// TwinCAT 3 PLC project Untitled1
// ProgramVersion: 3.1.4024.0
// libraries:
//   Tc2_HVAC, * (Beckhoff Automation GmbH)
//   Tc2_Standard, * (Beckhoff Automation GmbH)
//   Tc2_System, * (Beckhoff Automation GmbH)
//   Tc2_SystemC69xx, * (Beckhoff Automation GmbH)
//   Tc3_Module, * (Beckhoff Automation GmbH)
//   Util, * (System)
//   VisuSymbols,3.5.10.0,System
// project tree:
//   / GlobalTextList.TcGTLO, PlcTask.TcTTO, Visualization Manager.TcVMO (not stored)
//   GVLs/ GVL.TcGVL
//   POUs/FunctionBlocks/ Start_Stop.TcPOU, Trapizoidal.TcPOU
//   POUs/Functions/ ScaleOutput.TcPOU
//   POUs/ MAIN.TcPOU
//   POUs/Programs/ Motor_Control.TcPOU, ProgramSequence.TcPOU, Reset.TcPOU
//   VISUs/ Visualization.TcVIS
// real-time tasks:
//   TASK PlcTask: cycle T#10ms, priority 20, ADS port 350

CONFIGURATION Untitled1
    RESOURCE PLC ON TwinCAT3
        TASK PlcTask(INTERVAL := T#10ms, PRIORITY := 20);
        PROGRAM MAIN WITH PlcTask : MAIN;
    END_RESOURCE
END_CONFIGURATION

// ---- GVLs/GVL.TcGVL
{attribute 'qualified_only'}
VAR_GLOBAL
	(*Digital Input*)
	SART_STOP AT %IX0.0 : BOOL;		 	 (*To Start And To Stop System*)
	EM_STOP AT %IX0.1 : BOOL; 			 (*To Turn Power Of The System*)
	Conveyor2_Free AT %IX0.2 : BOOL;	 (*When The Conveyor2 is free*)
	Reset_Count AT %IX0.3 : BOOL;  		 (*Reset the Product counter value*)
	
	(*Analog Inputs*) (*Hiervoor vanwege gemak gebruik gemaakt van 0,1,3 normaal zou dit hogere waarde zijn wat uitgelezen wordt*)
	SensorInput AT %IW100 : INT;		 (*Noting=0 Red=1 Blue=2 Collor detection sensor*)

	(*Digital Output*)
	Motor1_State AT %QX10.0 : BOOL; 	 (*To indicate if the morot is on or of (1=on 0=of)*)
	Motor2_State AT %QX10.1 : BOOL;		 (*To indicate if the morot is on or of (1=on 0=of)*)
	
	(*Analog Output*)
	Motor1_Speed AT %QW200 : DINT;		 (*The Motor 1 Speed Output 0-65535*)
	Motor2_Speed AT %QW201 : DINT;		 (*The Motor 2 Speed Output 0-65535*)
	
	(*System Variables*)
	SystemState : INT; 					 (*System State 0=OFF 1=ON 2=EM_STOP*)	
	System_Start_Stop : BOOL;			 (*GVL Start/Stop variable 0=stop 1=start*)
	ProductA_Amount : INT;				 (*Amount of products counted*)
	ProductB_Amount : INT;				 (*Amount of products counted*)
	
	(*Motor Variables*)
	SetMotor1_Speed : INT;				 (*Set The Motor Speed in the program from hmi km/h*)
	SetMotor2_Speed : INT; 				 (*Set The Motor Speed in the program from hmi km/h*)
	CurrentMotor1_Speed : INT;			 (*The current speed after Trapizoidal function*)
	CurrentMotor2_Speed : INT;			 (*The current speed after Trapizoidal function*)
	Motor2_DirectionL : BOOL;			 (*Determine Motor direction*)
	Motor2_DirectionR : BOOL;			 (*Determine Motor direct*)

	

END_VAR

// ---- POUs/MAIN.TcPOU
PROGRAM MAIN
VAR
END_VAR

(*Calling Different Programs*)
Motor_Control ();
ProgramSequence ();
Reset ();

END_PROGRAM

// ---- POUs/Programs/Motor_Control.TcPOU
PROGRAM Motor_Control
VAR
	Start_Stop_0: Start_Stop;
	Trapizoidal_0: Trapizoidal;
	Trapizoidal_1: Trapizoidal;
	BLINK_0: BLINK;
	R_TRIG_0: R_TRIG;
	
	Timer : BOOL;
END_VAR

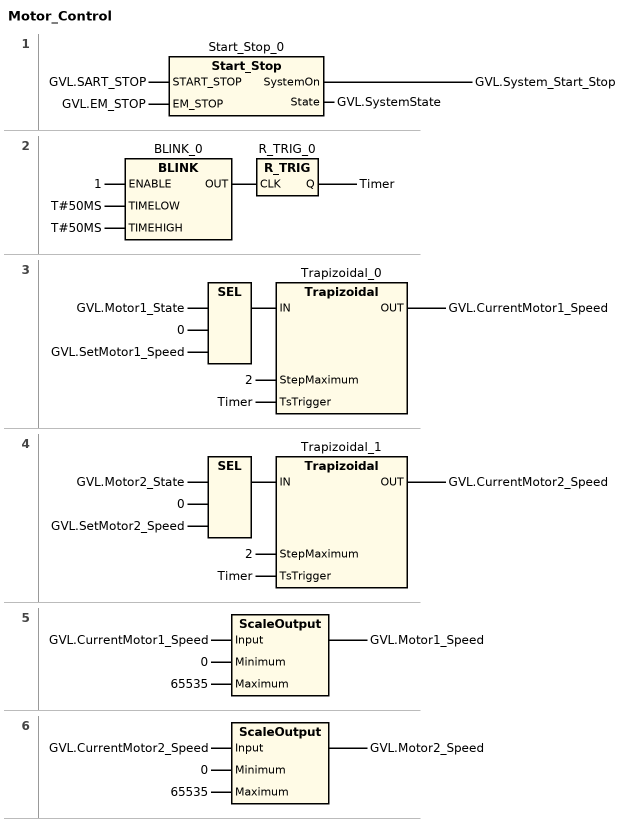
// NETWORK 1
Start_Stop_0(START_STOP := GVL.SART_STOP, EM_STOP := GVL.EM_STOP, State => GVL.SystemState); // Start_Stop
GVL.System_Start_Stop := Start_Stop_0.SystemOn;

// NETWORK 2
BLINK_0(ENABLE := 1, TIMELOW := T#50MS, TIMEHIGH := T#50MS); // BLINK
R_TRIG_0(CLK := BLINK_0.OUT); // R_TRIG
Timer := R_TRIG_0.Q;

// NETWORK 3
Trapizoidal_0(IN := SEL(GVL.Motor1_State, 0, GVL.SetMotor1_Speed), StepMaximum := 2, TsTrigger := Timer); // Trapizoidal
GVL.CurrentMotor1_Speed := Trapizoidal_0.OUT;

// NETWORK 4
Trapizoidal_1(IN := SEL(GVL.Motor2_State, 0, GVL.SetMotor2_Speed), StepMaximum := 2, TsTrigger := Timer); // Trapizoidal
GVL.CurrentMotor2_Speed := Trapizoidal_1.OUT;

// NETWORK 5
GVL.Motor1_Speed := ScaleOutput(Input := GVL.CurrentMotor1_Speed, Minimum := 0, Maximum := 65535);

// NETWORK 6
GVL.Motor2_Speed := ScaleOutput(Input := GVL.CurrentMotor2_Speed, Minimum := 0, Maximum := 65535);

END_PROGRAM

// ---- POUs/FunctionBlocks/Start_Stop.TcPOU
(*Vincent Molenkamp : 519540*)
FUNCTION_BLOCK Start_Stop
VAR_INPUT
	START_STOP : BOOL;
	EM_STOP : BOOL;
END_VAR
VAR_OUTPUT
	SystemOn : BOOL;
	State : INT;
END_VAR

VAR
	X: INT;
END_VAR

CASE X OF
	0: IF START_STOP THEN
		SystemOn := 1;
		X := 1;
		END_IF;
	1: IF NOT START_STOP THEN
			X := 2;
			State := 1;
		END_IF;
	2: IF START_STOP THEN
		SystemOn := 0;
		X := 3;
		END_IF;	
	3: IF NOT START_STOP THEN
		X := 0;	
		State := 0;
		END_IF;
	END_CASE
	
	IF NOT EM_STOP THEN
	X := 4;
	SystemOn := 0;
	State := 2;
	END_IF; 
	
	IF X = 4 AND EM_STOP AND NOT START_STOP THEN
		X := 0;
	END_IF

END_FUNCTION_BLOCK

// ---- POUs/FunctionBlocks/Trapizoidal.TcPOU
(*Vincent Molenkamp : 519540*)
FUNCTION_BLOCK Trapizoidal
(*Function Block To slowly increase speed*)
VAR_INPUT
	IN: INT;
	StepMaximum: INT;
	TsTrigger: BOOL;
END_VAR

VAR_OUTPUT	
	OUT: INT;
END_VAR

VAR
	Y_1: INT;
	Y_0: INT;
END_VAR

IF TsTrigger = 1 THEN
Y_1 := Y_0; (*De waarde van de vorige cicle in Y_1 Zetten*)

(*Wanneer de waarde van de voorige cicle lager is als de waarde van de nieuwe dan + 1 tot hij gelijk is*)
IF Y_1 < IN THEN
	Y_0 := 	Y_1 + StepMaximum;
END_IF

(*Wanneer de waarde van de voorige cicle Hoger is als de waarde van de nieuwe dan - 1 tot hij gelijk is*)
IF Y_1 > IN THEN
	Y_0 := Y_1 - StepMaximum;
END_IF

(*De output waarde meegeven*)
OUT := Y_0;
END_IF

END_FUNCTION_BLOCK

// ---- POUs/Functions/ScaleOutput.TcPOU
(*Vincent Molenkamp : 519540*)
FUNCTION ScaleOutput : DINT
(*Om de output waarde te scalen naar Van DINT naar WORD*)
VAR_INPUT	
	Input: INT;	  (*waarde die gescaled moet worden*)
	Minimum: INT; (*De minimum input waarde*)
	Maximum: INT; (*De maximum input waarde*)
END_VAR
VAR
	X: DINT;
END_VAR

(* To set minimum and maximum values for the input *)
IF Input < Minimum THEN
	Input := Minimum;
ELSIF Input > Maximum THEN
	Input := Maximum;
END_IF

(* Calculating the output value does not work with negative minimum *) 
ScaleOutput := ((Input-Minimum)*65535)/(Maximum-Minimum);

END_FUNCTION

// ---- POUs/Programs/ProgramSequence.TcPOU
PROGRAM ProgramSequence
VAR
	X: INT;
END_VAR

IF NOT GVL.System_Start_Stop THEN
	X := 10;
	GVL.Motor1_State := 0;
	GVL.Motor2_State := 0;	
END_IF

	CASE X OF
0: IF NOT GVL.Motor1_State THEN
 	GVL.Motor1_State := 1;
	X := 1;
	END_IF
	
1: IF GVL.SensorInput = 1 THEN
	GVL.Motor2_Direction := 0;
	GVL.Motor2_State := 1;
	GVL.ProductA_Amount := GVL.ProductA_Amount + 1;
	X := 2;
	ELSIF GVL.SensorInput = 2 THEN
	GVL.Motor2_Direction := 1;
	GVL.Motor2_State := 1;
	X := 2;
	GVL.ProductB_Amount := GVL.ProductB_Amount + 1;
	END_IF
	
2: 	GVL.Motor1_State := 0;
	IF GVL.Conveyor2_Free THEN
	X := 0;
	END_IF
	END_CASE

END_PROGRAM

// ---- POUs/Programs/Reset.TcPOU
PROGRAM Reset
(*What happens when reset is pressed*)
VAR
END_VAR

IF GVL.Reset_Count THEN
	GVL.ProductA_Amount := 0; (*To Reset Product Count*)
	GVL.ProductB_Amount := 0; (*To Reset Product Count*)
END_IF

END_PROGRAM

// ---- GlobalTextList.TcGTLO
TEXTLIST GlobalTextList
  21 = 'Amount A:%i'
  901 = 'Amount B:%i'
  356 = 'Conveyor 2 Free'
  483 = 'EM_Stop'
  0 = 'Motor 1'
  269 = 'Motor 1 Speed'
  816 = 'Motor 2'
  610 = 'Motor 2 Speed'
  52 = 'Product Type'
  237 = 'Reset Count'
  958 = 'Sensors'
  700 = 'Set Motor 1 Speed:%i'
  46 = 'Start/Stop'
  395 = 'Start_Stop Button'
  487 = 'System State:%i'
END_TEXTLIST

// ---- VISUs/Visualization.TcVIS
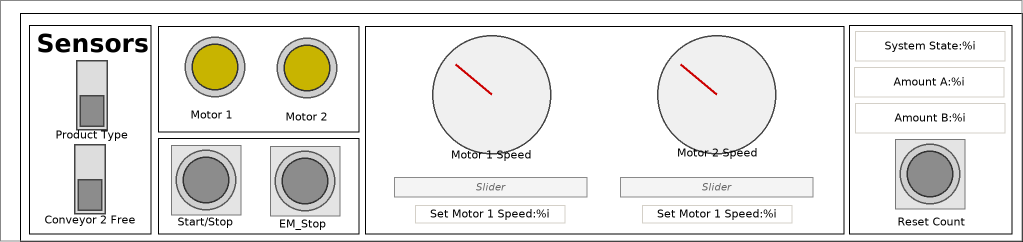
VISUALIZATION Visualization  // 1023x242
    Rectangle (20,13 1003x229)
    Rectangle (849,25 163x209)
    Rectangle (158,138 201x96)
    Rectangle (365,26 479x208)
    Rectangle (158,26 201x106)
    Rectangle (29,25 122x209)
    Lamp1 (180,32 70x70), style: Lamp-Lamp1-Yellow
    Lamp1 (272,33 70x70), variable: GVL.Motor2_State, style: Lamp-Lamp1-Yellow
    DipSwitch (57,60 70x70), variable: GVL.SensorInput, behaviour: TOGGLE, style: Switch-DipSwitch-Gray
    DipSwitch (55,144 70x70), variable: GVL.Conveyor2_Free, behaviour: TOGGLE, style: Switch-DipSwitch-Gray
    Label (18,28 150x30), "Sensors"
    Label (176,100 71x30), "Motor 1"
    Label (271,102 71x30), "Motor 2"
    Meter180 (386,35 211x119), value: GVL.CurrentMotor1_Speed, style: Meter-Meter180-Gray, scale format: %.1f, scale 0..100
    Meter180 (611,35 211x119), value: GVL.CurrentMotor2_Speed, style: Meter-Meter180-Gray, scale format: %.1f, scale 0..100
    Label (430,140 123x30), "Motor 1 Speed"
    Label (656,138 123x30), "Motor 2 Speed"
    Slider (394,177 193x20), variable: GVL.SetMotor1_Speed, scale 0..100
    Slider (620,177 193x20), variable: GVL.SetMotor2_Speed, scale 0..100
    PushSwitchLed (270,146 70x70), variable: GVL.EM_STOP, behaviour: TOGGLE, style: Switch-PushSwitchLed-Gray
    PushSwitch (171,145 70x70), variable: GVL.SART_STOP, behaviour: TOGGLE, style: Switch-PushSwitch-Gray
    Label (170,207 71x30), "Start/Stop"
    Label (267,209 71x30), "EM_Stop"
    Textfield (855,31 150x30), "System State:%i", text variable: GVL.SystemState
    Textfield (415,205 150x18), "Set Motor 1 Speed:%i", text variable: GVL.SetMotor1_Speed
    Textfield (642,205 150x18), "Set Motor 1 Speed:%i", text variable: GVL.SetMotor2_Speed
    Label (41,205 98x30), "Conveyor 2 Free"
    Label (43,120 98x30), "Product Type"
    Textfield (854,67 150x30), "Amount A:%i", text variable: GVL.ProductA_Amount
    Textfield (855,103 150x30), "Amount B:%i", text variable: GVL.ProductB_Amount
    PushSwitch (895,139 70x70), variable: GVL.Reset_Count, behaviour: TOGGLE, style: Switch-PushSwitch-Gray
    Label (870,207 123x30), "Reset Count"
END_VISUALIZATION
